TEXTLIST tlTransporterSequence_1
  0 = 'Initialization'
  5 = 'Back to normal state'
  10 = 'Wait for next cycle'
  12 = 'Waiting for parts entrace'
  14 = 'Waiting for parts going on carrdrige'
  16 = 'Allowing carrdrige move to chamber position'
  18 = 'Waiting for postition change of carrdrige'
  20 = 'Waiting for parts delivery to chamber'
  22 = 'Waiting for back to entry position'
  24 = 'Waiting for dors closed'
  25 = 'Waiting for end of cycle'
  26 = 'Waiting for dors opened'
  28 = 'Waiting for takeout position'
  30 = 'Unlocking carrdrige'
  32 = 'Locking Cardrige'
  34 = 'Opening exit lock'
  36 = 'Closing exit lock'
  90 = 'Error occur'
  91 = 'Wait for reset'
  95 = 'Performing reset sequence'
   = ''
END_TEXTLIST

(* stored: Version 1.1.0.1, ProductVersion 3.1.4024.13
   TextList tlTransporterSequence_1: Id {12bed802-f6d6-42fa-ac6e-1b39cea779b8} *)
